% RSLogix 500 project task2.RSS, saved by version 8.30.00.16 %
PROJECT "UNTITLED"    % processor: Bul.1763 MicroLogix 1100 Series B %

PROGRAM FILES
  LAD 2   4 rungs

DATA FILES
  O0 OUTPUT  4 elements
  I1 INPUT  6 elements
  S2 STATUS  66 elements
  B3 BINARY  1 elements
  T4 TIMER  3 elements
  C5 COUNTER  1 elements
  R6 CONTROL  1 elements
  N7 INTEGER  1 elements
  F8 FLOAT  1 elements

LADDER 2
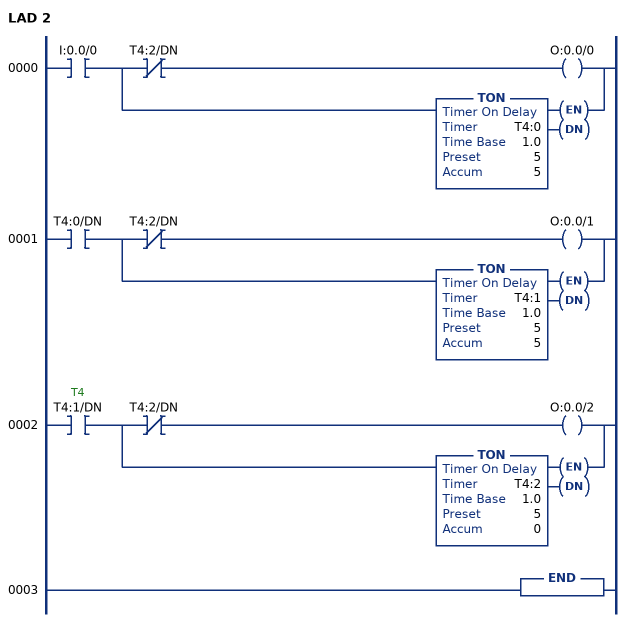
% Rung: 0 %
SOR XIC I:0.0/0 BST XIO T4:2/DN OTE O:0.0/0 NXB TON T4:0 1.0 5 5 BND EOR
% Rung: 1 %
SOR XIC T4:0/DN BST XIO T4:2/DN OTE O:0.0/1 NXB TON T4:1 1.0 5 5 BND EOR
% Rung: 2 %
SOR XIC T4:1/DN BST XIO T4:2/DN OTE O:0.0/2 NXB TON T4:2 1.0 5 0 BND EOR
%   T4:1/DN  T4 %
% Rung: 3 %
SOR END EOR

DATA TABLE (non-zero values as saved)
DATA T4
% .PRE .ACC %
% T4:0 % 5 5
% T4:1 % 5 5
% T4:2 % 5 0
